// TIA Portal V20 export
TYPE "type_emRelations_em3_cmStatus"
// stored: Access Published, Namespace Unit1
   STRUCT
      TopTapeJRDetect : "LBC_typeDigitalSignalControlNode";
      TopTapeDiameter : "LBC_typeDigitalSignalControlNode";
      TopTapeAxisX : "LBC_typeAxis64PosControlNode";
      TopTapeAxisY : "LBC_typeAxis64PosControlNode";
      TopTapeLoadingBwdFwd : "LBC_typeTwoWayActuatorControlNode";
      TopTapeLoadingClampOpenClose : "LBC_typeTwoWayActuatorControlNode";
      TopTapeCutterUpDown : "LBC_typeTwoWayActuatorControlNode";
      TopTapeCutterClampUpDown : "LBC_typeTwoWayActuatorControlNode";
      TopTapeTensionBwdFwd : "LBC_typeTwoWayActuatorControlNode";
      TopTapeAttachmentUpDown : "LBC_typeTwoWayActuatorControlNode";
      TopTapeClampTopLeftUpDown : "LBC_typeTwoWayActuatorControlNode";
      TopTapeClampTopCenterUpDown : "LBC_typeTwoWayActuatorControlNode";
      TopTapeClampTopRightUpDown : "LBC_typeTwoWayActuatorControlNode";
      TopTapeClampBtmDownUp : "LBC_typeTwoWayActuatorControlNode";
      TopTapeClampAllOpenClose : "LBC_typeTwoWayActuatorControlNode";
      TopTapeAttachmentVaccumOffOn : "LBC_typeTwoWayActuatorControlNode";
      QrHandyReader : "LER_typeDM8700ControlNode";
   END_STRUCT;
END_TYPE
